// TIA Portal V19 export
DATA_BLOCK "CoilHandlingMatCounter_PERS"   // DB193
{ DB_Accessible_From_OPC_UA := 'FALSE' }
// stored: DBAccessibleFromOPCUA false, MemoryReserve 100
   VAR RETAIN
      PersistentValues : "MatCountPersistent";
   END_VAR
BEGIN
   PersistentValues.Data.AxPosition := 0.0;
   PersistentValues.Data.AxPositionPrevious := 0.0;
   PersistentValues.Data.FAK := 0.0;
   PersistentValues.Data.CounterValueInit := 0.0;
   PersistentValues.Data.CounterOffset := 0.0;
   PersistentValues.Data.CounterValue := 0.0;
   PersistentValues.Data.FAKPrevious := 0.0;
   PersistentValues.Data.AX_MODULE := 0.0;
   PersistentValues.Data.COUNTER_MODULE := 0.0;
   PersistentValues.Par.FAK := 1.0010982162041;
END_DATA_BLOCK
